screen "main" 1920x1080, template "Template_1"
   TextField "Static Text47_8" at 798,552 size 36x17; Text 'TE1.3 / TE04.1'
   Group "Group_10" at 795,569 size 82x26
   SymbolLibrary "Symbol library_115" at 1565,119 size 14x20
      Visibility <- "Di_1Ga01"
      Appearance <- "ViewLine_DB_Line24"
   SymbolLibrary "Symbol library_114" at 1552,129 size 27x27
      Visibility <- "Di_1Ga01"
      Appearance <- "ViewLine_DB_Line24"
   SymbolLibrary "Symbol library_113" at 1520,142 size 34x14
      Visibility <- "Di_1Ga01"
      Appearance <- "ViewLine_DB_Line24"
   SymbolLibrary "Symbol library_116" at 1565,120 size 14x57
      Visibility <- "Di_1Ga02"
      Appearance <- "ViewLine_DB_Line25"
   SymbolLibrary "Symbol library_117" at 1552,167 size 27x27
      Visibility <- "Di_1Ga02"
      Appearance <- "ViewLine_DB_Line25"
   SymbolLibrary "Symbol library_118" at 1520,180 size 34x14
      Visibility <- "Di_1Ga02"
      Appearance <- "ViewLine_DB_Line25"
   Rectangle "Rectangle_1r" at 50,206 size 75x24; ToolTipText 'Температура НС'
   TextField "Text field_1asd" at 100,206 size 19x22; Text 'С°'
   IOField "IO Field_10" at 43,204 size 56x26; FormatPattern 999.9
      ProcessValue <- "AiCh_TE7.1_Px"
   Rectangle "Rectangle_2cxv" at 182,511 size 75x24; ToolTipText 'Температура НС'
   TextField "Text field_3df" at 232,511 size 19x22; Text 'С°'
   IOField "IO Field_1" at 175,509 size 56x26; FormatPattern 999.9
      ProcessValue <- "AiCh_TE7.2_Px"
   Rectangle "Rectangle_3dcxf" at 920,570 size 75x24; ToolTipText 'Температура НС'
   TextField "Text field_4ыва" at 970,570 size 19x22; Text 'С°'
   IOField "IO Field_2" at 913,568 size 56x26; FormatPattern 999.9
      ProcessValue <- "AiCh_TE1.1_Px"
   Rectangle "Rectangle_4" at 921,495 size 68x24; ToolTipText 'Температура НС'
   TextField "Text field_6ret" at 962,495 size 18x22; Text '%'
   IOField "IO Field_3" at 924,493 size 36x26; FormatPattern 999
      ProcessValue <- "AiCh_LIC1.1_Px"
   Rectangle "Rectangle_5" at 802,571 size 75x24; ToolTipText 'Температура НС'
   IOField "IO Field_4" at 795,569 size 56x26; FormatPattern 999.9
      ProcessValue <- "AiCh_TE1.3_Px"
   TextField "Text field_8qw" at 852,571 size 19x22; Text 'С°'
   Rectangle "Rectangle_6" at 804,342 size 75x24; ToolTipText 'Температура НС'
   IOField "IO Field_5" at 797,340 size 56x26; FormatPattern 999.9
      ProcessValue <- "AiCh_TE1.2_Px"
   TextField "Text field_9x" at 854,342 size 19x22; Text 'С°'
   Rectangle "Rectangle_8" at 1342,495 size 68x24; ToolTipText 'Температура НС'
   TextField "Text field_11as" at 1383,495 size 18x22; Text '%'
   IOField "IO Field_6" at 1345,493 size 36x26; FormatPattern 999
      ProcessValue <- "AiCh_LIC2.1_Px"
   Rectangle "Rectangle_9" at 1341,570 size 75x24; ToolTipText 'Температура НС'
   TextField "Text field_12ew" at 1391,570 size 19x22; Text 'С°'
   IOField "IO Field_7" at 1334,568 size 56x26; FormatPattern 999.9
      ProcessValue <- "AiCh_TE2.1_Px"
   TextField "Static Text47_5" at 1219,547 size 36x17; Text 'TE2.3 / TE04.1'
   Group "Group_12" at 1216,564 size 82x26
   Rectangle "Rectangle_10" at 1223,566 size 75x24; ToolTipText 'Температура НС'
   IOField "IO Field_8" at 1216,564 size 56x26; FormatPattern 999.9
      ProcessValue <- "AiCh_TE2.3_Px"
   TextField "Text field_13azq" at 1273,566 size 19x22; Text 'С°'
   Group "Group_14" at 797,340 size 82x26
   TextField "Static Text47_7" at 820,324 size 36x17; Text 'TE1.2 / TE04.1'
   Rectangle "Rectangle_11" at 1225,342 size 75x24; ToolTipText 'Температура НС'
   IOField "IO Field_9" at 1218,340 size 56x26; FormatPattern 999.9
      ProcessValue <- "AiCh_TE2.2_Px"
   TextField "Text field_14ty" at 1275,342 size 19x22; Text 'С°'
   Group "Group_16" at 1218,340 size 82x26
   TextField "Static Text47_10" at 1241,324 size 36x17; Text 'TE2.2 / TE04.1'
   Rectangle "Rectangle_12" at 230,351 size 68x24; ToolTipText 'Температура НС'
   TextField "Text field_15fd" at 271,351 size 18x22; Text '%'
   IOField "IO Field_11" at 233,349 size 36x26; FormatPattern 999
      ProcessValue <- "Data.LevelVO"
   IOField "I/O field_2" at 165,649 size 39x20; FormatPattern 999
      ProcessValue <- "Data_Reg_01RV01_LMN"
   TextField "Text field_16d" at 201,650 size 19x19; Text '%'
   IOField "I/O field_1" at 309,929 size 39x20; FormatPattern 999
      ProcessValue <- "DriveM7_1.Vx"
   TextField "Text field_17zzz" at 345,930 size 19x19; Text '%'
   IOField "I/O field_3" at 562,932 size 39x20; FormatPattern 999
      ProcessValue <- "DriveM7_2.Vx"
   TextField "Text field_18" at 598,933 size 19x19; Text '%'
   IOField "I/O field_4" at 921,245 size 43x20; FormatPattern s999
      ProcessValue <- "DriveM1_1.Vx"
   TextField "Text field_19" at 965,246 size 19x19; Text '%'
   IOField "I/O field_6" at 1342,245 size 43x20; FormatPattern s999
      ProcessValue <- "DriveM2_1.Vx"
   TextField "Text field_21" at 1386,246 size 19x19; Text '%'
   Rectangle "Rectangle_13" at 182,487 size 75x24; ToolTipText 'Температура НС'
   TextField "Text field_20" at 232,487 size 19x22; Text 'С°'
   IOField "IO Field_17" at 175,485 size 56x26; FormatPattern 999.9
      ProcessValue <- "Data_Reg_01RV01_Sp"
   Rectangle "Rectangle_14" at 920,546 size 75x24; ToolTipText 'Температура НС'
   TextField "Text field_22" at 970,546 size 19x22; Text 'С°'
   IOField "IO Field_18" at 913,544 size 56x26; FormatPattern 999.9
      ProcessValue <- "Data_Reg_TE1_1_Sp"
   Rectangle "Rectangle_15" at 230,327 size 68x24; ToolTipText 'Температура НС'
   TextField "Text field_23" at 271,327 size 18x22; Text '%'
   IOField "IO Field_19" at 233,325 size 36x26; FormatPattern 999
      ProcessValue <- "Data_Reg_M7_1_Sp"
   Rectangle "Rectangle_16" at 1341,546 size 75x24; ToolTipText 'Температура НС'
   TextField "Text field_24" at 1391,546 size 19x22; Text 'С°'
   IOField "IO Field_20" at 1334,544 size 56x26; FormatPattern 999.9
      ProcessValue <- "Data_Reg_TE2_1_Sp"
   SymbolLibrary "Symbol library_130" at 703,869 size 202x14
      Appearance <- "ViewLine_DB_Line23"
   SymbolLibrary "Symbol library_15" at 917,869 size 415x14
      Appearance <- "ViewLine_DB_Line18"
   SymbolLibrary "Symbol library_49" at 1379,706 size 111x13
      Appearance <- "ViewLine_DB_Line17"
   SymbolLibrary "Symbol library_3" at 861,370 size 31x13
      Appearance <- "ViewLine_DB_Line11"
   SymbolLibrary "Symbol library_45" at 959,706 size 111x13
      Appearance <- "ViewLine_DB_Line13"
   SymbolLibrary "Symbol library_106" at 345,501 size 12x113
      Appearance <- "ViewLine_DB_Line7"
   SymbolLibrary "Symbol library_82" at 289,819 size 14x38
      Appearance <- "ViewLine_DB_Line3"
   SymbolLibrary "Symbol library_16" at 260,444 size 14x436
      Appearance <- "ViewLine_DB_Line1"
   SymbolLibrary "Symbol library_156" at 569,331 size 25x25
      Appearance <- "DrvCell_M3_Km1"
   SymbolLibrary "Symbol library_157" at 460,326 size 53x13
      Appearance <- "DrvCell_M3_Km1"
   ScreenModuleView "M_3_1" at 511,323 size 60x51; ScreenModuleType ""
      Guid_{11997190-24475} <- "DrvCell_M3_Err"
      Guid_{11997190-24471} <- "DrvCell_M3_Km1"
   Button "Button_4ert" at 510,323 size 61x52; TextOff 'Text'
      on Press: function_b14e0dd5("DrvCell_M3_SB1", 0)
   SymbolLibrary "Symbol library_44" at 949,604 size 14x235
      Appearance <- "ViewLine_DB_Line10"
   SymbolLibrary "Symbol library_66" at 885,598 size 25x25
      Appearance <- "ViewLine_DB_Line11"
   GraphicView "Graphic view_5" at 872,330 size 164x288; Picture "Graphic_1"
   SymbolLibrary "Symbol library_39" at 552,854 size 12x25
      Appearance <- "ViewLine_DB_Line4"
   SymbolLibrary "Symbol library_21" at 365,499 size 12x64
      Appearance <- "ViewLine_DB_Line6"
   SymbolLibrary "Symbol library_80" at 1586,695 size 96x14
      Appearance <- "ViewLine_DB_Line21"
   SymbolLibrary "Symbol library_14" at 214,202 size 25x25
      Appearance <- "ViewLine_DB_Line2"
   SymbolLibrary "Symbol library_10" at 153,224 size 13x158
      Appearance <- "ViewLine_DB_Line2"
   SymbolLibrary "Symbol library_47" at 107,377 size 125x14
      Appearance <- "ViewLine_DB_Line1"
   SymbolLibrary "Symbol library_5" at 218,206 size 98x241
   Bar "Bar_5" at 224,244 size 86x168; MinimumValue 0; MaximumValue 100
      ProcessValue <- "Data.LevelVO"
   SymbolLibrary "Symbol library_71" at 1306,598 size 25x25
      Appearance <- "ViewLine_DB_Line15"
   SymbolLibrary "Symbol library_56" at 1282,370 size 31x13
      Appearance <- "ViewLine_DB_Line15"
   SymbolLibrary "Symbol library_9" at 1369,604 size 14x235
      Appearance <- "ViewLine_DB_Line14"
   GraphicView "Graphic view_1" at 1293,330 size 164x288; Picture "Graphic_1"
   Bar "Bar_1" at 1314,352 size 124x243; MinimumValue 0; MaximumValue 100
      ProcessValue <- "AiCh_LIC2.1_Px"
   Bar "Bar_2" at 893,352 size 124x243; MinimumValue 0; MaximumValue 100
      ProcessValue <- "AiCh_LIC1.1_Px"
   SymbolLibrary "Symbol library_110" at 968,800 size 395x14
      Appearance <- "ViewLine_DB_Line3"
   SymbolLibrary "Symbol library_53" at 32,131 size 14x237
      Appearance <- "ViewLine_DB_Line1"
   SymbolLibrary "Symbol library_11" at 177,202 size 47x13
      Appearance <- "ViewLine_DB_Line2"
   SymbolLibrary "Symbol library_58" at 28,105 size 21x41
   SymbolLibrary "Symbol library_23" at 381,476 size 104x12
      Appearance <- "ViewLine_DB_Line5"
   SymbolLibrary "Symbol library_25" at 492,495 size 12x189
      Appearance <- "ViewLine_DB_Line5"
   SymbolLibrary "Symbol library_79" at 381,440 size 140x12
      Appearance <- "ViewLine_DB_Line4"
   SymbolLibrary "Symbol library_6" at 253,150 size 54x59
   SymbolLibrary "Symbol library_7" at 303,150 size 65x30
   SymbolLibrary "Symbol library_158" at 581,299 size 13x35
      Appearance <- "DrvCell_M3_Km1"
   SymbolLibrary "Symbol library_160" at 578,147 size 13x58
   SymbolLibrary "Symbol library_31" at 284,885 size 31x16
   SymbolLibrary "Symbol library_36" at 1335,869 size 156x14
      Appearance <- "ViewLine_DB_Line19"
   SymbolLibrary "Symbol library_12" at 153,202 size 25x25
      Appearance <- "ViewLine_DB_Line2"
   TextField "Text field_2fdsa" at 314,702 size 19x34; Text 'Y'
   SymbolLibrary "Symbol library_186" at 678,132 size 14x727
      Appearance <- "ViewLine_DB_Line23"
   SymbolLibrary "Symbol library_41" at 271,906 size 15x15
      Appearance <- "ViewLine_DB_Line8"
   SymbolLibrary "Symbol library_46" at 168,934 size 99x8
      Appearance <- "ViewLine_DB_Line8"
   SymbolLibrary "Symbol library_43" at 146,930 size 30x15
   SymbolLibrary "Symbol library_48" at 264,927 size 15x15
      Appearance <- "ViewLine_DB_Line8"
   SymbolLibrary "Symbol library_50" at 271,914 size 8x16
      Appearance <- "ViewLine_DB_Line8"
   SymbolLibrary "Symbol library_95" at 678,107 size 27x27
      Appearance <- "ViewLine_DB_Line23"
   SymbolLibrary "Symbol library_91" at 1012,142 size 503x14
      Appearance <- "ViewLine_DB_Line24"
   SymbolLibrary "Symbol library_90" at 693,107 size 824x14
      Appearance <- "ViewLine_DB_Line23"
   SymbolLibrary "Symbol library_93" at 1439,180 size 78x14
      Appearance <- "ViewLine_DB_Line25"
   SymbolLibrary "Symbol library_98" at 1577,107 size 293x14
      Appearance <- "ViewLine_DB_Line22"
   SymbolLibrary "Symbol library_99" at 574,121 size 21x41
   SymbolLibrary "Symbol library_100" at 442,321 size 41x21
   SymbolLibrary "Symbol library_108" at 1590,546 size 95x14
      Appearance <- "ViewLine_DB_Line20"
   SymbolLibrary "Symbol library_109" at 1672,542 size 41x21
   SymbolLibrary "Symbol library_107" at 313,800 size 211x14
      Appearance <- "ViewLine_DB_Line3"
   SymbolLibrary "Symbol library_111" at 1388,800 size 105x14
      Appearance <- "ViewLine_DB_Line3"
   SymbolLibrary "Symbol library_105" at 1479,796 size 41x21
   TextField "Static Text47_2" at 199,470 size 33x16; Text 'TE7.2 / TE04.1'
   SymbolLibrary "Symbol library_29" at 695,800 size 247x14
      Appearance <- "ViewLine_DB_Line3"
   Circle "Circle_23" at 1030,351 size 25x25
      Appearance <- "Di_Lah1.1"
   SymbolLibrary "Symbol library_57" at 944,610 size 37x48
   TextField "Static Text47_6" at 938,530 size 33x16; Text 'TE1.1 / TE04.1'
   TextField "Static Text47_9" at 935,479 size 40x16; Text 'LIC 1.1 / TE04.1'
   SymbolLibrary "Symbol library_123" at 989,168 size 14x209
      Appearance <- "ViewLine_DB_Line24"
   SymbolLibrary "Symbol library_55" at 989,142 size 27x27
      Appearance <- "ViewLine_DB_Line24"
   SymbolLibrary "Symbol library_96" at 1415,180 size 27x27
      Appearance <- "ViewLine_DB_Line25"
   SymbolLibrary "Symbol library_97" at 678,856 size 27x27
      Appearance <- "ViewLine_DB_Line23"
   SymbolLibrary "Symbol library_83" at 289,800 size 27x27
      Appearance <- "ViewLine_DB_Line3"
   SymbolLibrary "Symbol library_18" at 260,874 size 27x27
      Appearance <- "ViewLine_DB_Line1"
   SymbolLibrary "Symbol library_54" at 32,364 size 27x27
      Appearance <- "ViewLine_DB_Line1"
   SymbolLibrary "Symbol library_24" at 480,476 size 24x22
      Appearance <- "ViewLine_DB_Line5"
   GraphicView "Graphic view_4" at 526,196 size 122x112; Picture "Graphic_5"
   Circle "Circle_26" at 617,208 size 25x25
      Appearance <- "Di_Lah01"
   Circle "Circle_15" at 617,271 size 25x25
      Appearance <- "Di_Lal01"
   Line "Line_3" at 913,810 size 42x26
      Visibility <- "Di_Ga1.1"
   Line "Line_5" at 1333,810 size 42x26
      Visibility <- "Di_Ga2.1"
   Line "Line_1" at 913,838 size 42x36
      Visibility <- "Di_Ga1.2"
   Line "Line_6" at 1333,838 size 42x36
      Visibility <- "Di_Ga2.2"
   SymbolLibrary "Symbol library_94" at 1516,107 size 50x14
      Visibility <- "Di_1Ga06"
      Appearance <- "ViewLine_DB_Line23"
   Group "Group_2" at 1520,119 size 59x37
      Visibility <- "Di_1Ga01"
   Group "Group_3" at 1520,120 size 59x74
      Visibility <- "Di_1Ga02"
   ScreenModuleView "V7_31_2" at 76,350 size 50x42; ScreenModuleType ""
      Guid_{11997190-20001} <- "DrvCell_V7_3_Err"
      Guid_{11997190-19997} <- "DrvCell_V7_3_Km1"
   TextField "Static Text47_1" at 68,190 size 33x16; Text 'TE7.1 / TE04.1'
   Group "Group_17" at 43,204 size 82x26; FormatPattern 999.9
   Group "Group_1" at 175,509 size 82x26; FormatPattern 999.9
   ScreenModuleView "M7_1_1" at 283,856 size 88x65; ScreenModuleType ""
      Guid_{11997190-20935} <- "DrvCell_M7_1_Km1"
      Guid_{11997190-20939} <- "DrvCell_M7_1_Err"
   ScreenModuleView "M1_2_3" at 1480,850 size 60x51; ScreenModuleType ""
      Guid_{11997190-21672} <- "DrvCell_M5_Err"
      Guid_{11997190-21676} <- "DrvCell_M5_Km1"
   SymbolLibrary "Symbol library_17" at 910,338 size 88x135
   ScreenModuleView "M1_1_1" at 923,270 size 53x69; ScreenModuleType ""
      Guid_{11997190-22971} <- "DrvCell_M1_1_Err"
      Guid_{11997190-22975} <- "DrvCell_M1_1_Km1"
   SymbolLibrary "Symbol library_13" at 1364,610 size 37x48
   SymbolLibrary "Symbol library_92" at 1415,202 size 14x173
      Appearance <- "ViewLine_DB_Line25"
   SymbolLibrary "Symbol library_33" at 1333,338 size 88x135
   ScreenModuleView "M1_1_2" at 1347,270 size 53x69; ScreenModuleType ""
      Guid_{11997190-22971} <- "DrvCell_M2_1_Err"
      Guid_{11997190-22975} <- "DrvCell_M2_1_Km1"
   TextField "Text field_10v" at 1308,367 size 55x39; Text '№2'
   ScreenModuleView "V1_7_1" at 992,696 size 35x26; ScreenModuleType ""
      Guid_{11997190-23352} <- "DrvCell_V1_7_Err"
      Guid_{11997190-23356} <- "DrvCell_V1_7_Km1"
   Group "Group_6" at 921,493 size 68x26
   Group "Group_7" at 913,568 size 82x26
   TextField "Static Text47_3" at 1359,530 size 33x16; Text 'TE2.1 / TE04.1'
   TextField "Static Text47_4" at 1356,479 size 40x16; Text 'LIC 2.1 / TE04.1'
   Group "Group_8" at 1342,493 size 68x26
   Group "Group_9" at 1334,568 size 82x26
   Circle "Circle_3" at 1451,352 size 25x25
      Appearance <- "Di_Lah2.1"
   SymbolLibrary "Symbol library_67" at 838,370 size 25x25
      Appearance <- "ViewLine_DB_Line11"
   SymbolLibrary "Symbol library_147" at 814,390 size 25x25
      Appearance <- "ViewLine_DB_Line11"
   SymbolLibrary "Symbol library_102" at 814,413 size 13x26
      Appearance <- "ViewLine_DB_Line11"
   SymbolLibrary "Symbol library_64" at 838,393 size 13x257
      Appearance <- "ViewLine_DB_Line11"
   SymbolLibrary "Symbol library_65" at 906,610 size 25x25
      Appearance <- "ViewLine_DB_Line11"
   SymbolLibrary "Symbol library_63" at 906,622 size 25x25
      Appearance <- "ViewLine_DB_Line11"
   SymbolLibrary "Symbol library_59" at 738,649 size 114x13
      Appearance <- "ViewLine_DB_Line12"
   SymbolLibrary "Symbol library_68" at 708,645 size 41x21
   ScreenModuleView "V7_31_1" at 772,621 size 50x42; ScreenModuleType ""
      Guid_{11997190-20001} <- "DrvCell_V1_1_Err"
      Guid_{11997190-19997} <- "DrvCell_V1_1_Km1"
   SymbolLibrary "Symbol library_101" at 810,422 size 21x41
   SymbolLibrary "Symbol library_60" at 1259,370 size 25x25
      Appearance <- "ViewLine_DB_Line15"
   SymbolLibrary "Symbol library_61" at 1235,390 size 25x25
      Appearance <- "ViewLine_DB_Line15"
   SymbolLibrary "Symbol library_69" at 1235,413 size 13x26
      Appearance <- "ViewLine_DB_Line15"
   SymbolLibrary "Symbol library_70" at 1259,393 size 13x257
      Appearance <- "ViewLine_DB_Line15"
   SymbolLibrary "Symbol library_73" at 1327,610 size 25x25
      Appearance <- "ViewLine_DB_Line15"
   SymbolLibrary "Symbol library_74" at 1327,622 size 25x25
      Appearance <- "ViewLine_DB_Line15"
   SymbolLibrary "Symbol library_75" at 1159,649 size 114x13
      Appearance <- "ViewLine_DB_Line16"
   SymbolLibrary "Symbol library_76" at 1129,645 size 41x21
   SymbolLibrary "Symbol library_62" at 1231,422 size 21x41
   ScreenModuleView "V7_31_3" at 1196,621 size 50x42; ScreenModuleType ""
      Guid_{11997190-20001} <- "DrvCell_V2_1_Err"
      Guid_{11997190-19997} <- "DrvCell_V2_1_Km1"
   ScreenModuleView "V1_7_2" at 1412,696 size 35x26; ScreenModuleType ""
      Guid_{11997190-23352} <- "DrvCell_V2_7_Err"
      Guid_{11997190-23356} <- "DrvCell_V2_7_Km1"
   Group "Group_19" at 230,349 size 68x26
   ScreenModuleView "V1_7_3" at 198,923 size 35x26; ScreenModuleType ""
      Guid_{11997190-23352} <- "DrvCell_V7_1_Err"
      Guid_{11997190-23356} <- "DrvCell_V7_1_Km1"
   TextField "Static Text47_11" at 82,330 size 26x16; Text 'V7.3 / TE04.1'
   TextField "Static Text47_12" at 179,234 size 26x16; Text 'V7.4 / TE04.1'
   Button "Button_1yt" at 75,350 size 52x43; TextOff 'Text'
      on Press: function_b14e0dd5("DrvCell_V7_3_SB1", 0)
   SymbolLibrary "Symbol library_42" at 441,695 size 52x12
      Appearance <- "ViewLine_DB_Line5"
   SymbolLibrary "Symbol library_30" at 339,679 size 45x12
      Appearance <- "ViewLine_DB_Line5"
   ScreenModuleView "M_3_2" at 382,676 size 60x51; ScreenModuleType ""
      Guid_{11997190-24471} <- "DrvCell_M10_Km1"
      Guid_{11997190-24475} <- "DrvCell_M10_Err"
   SymbolLibrary "Symbol library_27" at 528,459 size 12x422
      Appearance <- "ViewLine_DB_Line4"
   SymbolLibrary "Symbol library_1" at 481,683 size 23x24
      Appearance <- "ViewLine_DB_Line5"
   SymbolLibrary "Symbol library_22" at 516,440 size 24x22
      Appearance <- "ViewLine_DB_Line4"
   SymbolLibrary "Symbol library_34" at 528,875 size 23x23
      Appearance <- "ViewLine_DB_Line4"
   SymbolLibrary "Symbol library_40" at 318,679 size 23x23
      Appearance <- "ViewLine_DB_Line5"
   TextField "adasd" at 650,858 size 19x34; Text 'Y'
   TextField "Static Text47_13" at 393,659 size 24x16; Text 'M10 / TE04.1'
   Button "Button_3fdg" at 382,676 size 60x52; TextOff 'Text'
      on Press: function_b14e0dd5("DrvCell_M10_SB1", 0)
   TextField "Static Text47_14" at 526,306 size 17x16; Text 'M3 / TE04.1'
   SymbolLibrary "Symbol library_2" at 361,550 size 21x41
   SymbolLibrary "Symbol library_19" at 643,834 size 23x23
      Appearance <- "ViewLine_DB_Line4"
   SymbolLibrary "Symbol library_20" at 573,834 size 76x12
      Appearance <- "ViewLine_DB_Line4"
   SymbolLibrary "Symbol library_26" at 552,834 size 23x23
      Appearance <- "ViewLine_DB_Line4"
   SymbolLibrary "Symbol library_28" at 533,912 size 8x22
      Appearance <- "ViewLine_DB_Line9"
   SymbolLibrary "Symbol library_32" at 526,927 size 15x15
      Appearance <- "ViewLine_DB_Line9"
   SymbolLibrary "Symbol library_37" at 533,899 size 15x15
      Appearance <- "ViewLine_DB_Line9"
   SymbolLibrary "Symbol library_38" at 444,934 size 87x8
      Appearance <- "ViewLine_DB_Line9"
   ScreenModuleView "V1_7_4" at 473,923 size 35x26; ScreenModuleType ""
      Guid_{11997190-23352} <- "DrvCell_V7_2_Err"
      Guid_{11997190-23356} <- "DrvCell_V7_2_Km1"
   TextField "Static Text58_1" at 9,65 size 62x32; Text 'Продукт, CIP+2 RV01'
   TextField "Static Text58_3" at 1474,770 size 35x16; Text 'CIP-2 / RV01'
   TextField "Static Text58_5" at 1716,535 size 62x32; Text 'Продукт, CIP+1 RV01'
   TextField "Static Text47_15" at 328,854 size 28x16; Text 'M7.1 / TE04.1'
   TextField "Static Text47_16" at 577,856 size 28x16; Text 'M7.2 / TE04.1'
   TextField "Static Text47_17" at 202,902 size 26x16; Text 'V7.1 / TE04.1'
   TextField "Static Text47_18" at 777,602 size 26x16; Text 'V1.1 / TE04.1'
   TextField "Static Text47_19" at 855,609 size 28x16; Text 'M1.2 / TE04.1'
   TextField "Static Text47_20" at 995,677 size 26x16; Text 'V1.7 / TE04.1'
   TextField "Static Text47_21" at 935,228 size 28x16; Text 'M1.1 / TE04.1'
   TextField "Static Text47_22" at 1359,228 size 28x16; Text 'M2.1 / TE04.1'
   TextField "Static Text47_23" at 1200,602 size 26x16; Text 'V2.1 / TE04.1'
   TextField "Static Text47_24" at 1276,609 size 28x16; Text 'M2.2 / TE04.1'
   TextField "Static Text47_25" at 1416,677 size 26x16; Text 'V2.7 / TE04.1'
   Button "Button_15" at 1398,684 size 65x49; TextOff 'Text'
      on Press: function_b14e0dd5("DrvCell_V2_7_SB1", 0)
   TextField "Static Text47_26" at 477,904 size 26x16; Text 'V7.2 / TE04.1'
   TextField "Static Text47_27" at 1785,887 size 17x16; Text 'M4 / TE04.1'
   TextField "Text field_7fd" at 885,367 size 55x39; Text '№1'
   Group "Group_11" at 795,552 size 82x43
   Group "Group_15" at 797,324 size 82x42
   Group "Group_18" at 1218,324 size 82x42
   Group "Group_13" at 1216,547 size 82x43; Text 'TE1.3'
   TextField "Static Text58_6" at 554,230 size 67x32; Text 'Ледянная вода RV01'
   TextField "Static Text58_7" at 81,922 size 61x32; Text 'Вода питьевая RV01'
   SymbolLibrary "Symbol library_35" at 1575,566 size 14x288
      Appearance <- "ViewLine_DB_Line20"
   SymbolLibrary "Symbol library_72" at 1540,853 size 35x14
      Appearance <- "ViewLine_DB_Line20"
   SymbolLibrary "Symbol library_77" at 1562,840 size 27x27
      Appearance <- "ViewLine_DB_Line20"
   SymbolLibrary "Symbol library_78" at 1575,546 size 27x27
      Appearance <- "ViewLine_DB_Line20"
   SymbolLibrary "Symbol library_81" at 1690,708 size 14x66
      Appearance <- "ViewLine_DB_Line21"
   SymbolLibrary "Symbol library_84" at 1677,695 size 27x27
      Appearance <- "ViewLine_DB_Line21"
   SymbolLibrary "Symbol library_85" at 1690,865 size 14x50
      Appearance <- "ViewLine_DB_Line21"
   SymbolLibrary "Symbol library_86" at 1707,926 size 55x14
      Appearance <- "ViewLine_DB_Line21"
   SymbolLibrary "Symbol library_87" at 1690,913 size 27x27
      Appearance <- "ViewLine_DB_Line21"
   GraphicView "Graphic view_2" at 1636,758 size 122x112; Picture "Graphic_5"
   TextField "Static Text58_4" at 1687,789 size 21x32; Text 'CIP ББ RV01'
   SymbolLibrary "Symbol library_88" at 1869,123 size 14x788
      Appearance <- "ViewLine_DB_Line22"
   SymbolLibrary "Symbol library_89" at 1818,910 size 48x14
      Appearance <- "ViewLine_DB_Line22"
   SymbolLibrary "Symbol library_103" at 1856,897 size 27x27
      Appearance <- "ViewLine_DB_Line22"
   SymbolLibrary "Symbol library_51" at 1856,107 size 27x27
      Appearance <- "ViewLine_DB_Line22"
   TextField "Static Text47_28" at 1503,830 size 17x16; Text 'M5 / TE04.1'
   ScreenModuleView "M1_2_4" at 1759,906 size 60x51; ScreenModuleType ""
      Guid_{11997190-21672} <- "DrvCell_M4_Err"
      Guid_{11997190-21676} <- "DrvCell_M4_Km1"
   SymbolLibrary "Symbol library_104" at 543,800 size 131x14
      Appearance <- "ViewLine_DB_Line3"
   SymbolLibrary "Symbol library_112" at 277,624 size 63x12
      Appearance <- "ViewLine_DB_Line7"
   SymbolLibrary "Symbol library_119" at 128,625 size 128x12
      Appearance <- "ViewLine_DB_Line7"
   SymbolLibrary "Symbol library_120" at 334,612 size 23x24
      Appearance <- "ViewLine_DB_Line7"
   SymbolLibrary "Symbol library_121" at 107,638 size 12x105
      Appearance <- "ViewLine_DB_Line7"
   SymbolLibrary "Symbol library_122" at 107,625 size 22x22
      Appearance <- "ViewLine_DB_Line7"
   SymbolLibrary "Symbol library_124" at 102,736 size 21x41
   Group "Group_20" at 165,649 size 55x20; FormatPattern 999
   Group "Group_21" at 309,929 size 55x20; FormatPattern 999
   Group "Group_22" at 562,932 size 55x20; FormatPattern 999
   Group "Group_23" at 921,245 size 63x20; FormatPattern 999
   Group "Group_25" at 1342,245 size 63x20; FormatPattern 999
   SymbolLibrary "Symbol library_127" at 1298,286 size 41x32
      Visibility <- "Data_Mixer2_Direction"
   SymbolLibrary "Symbol library_128" at 1414,286 size 41x32
      Visibility <- "Data_Mixer2_Direction"
   TextField "Text field_68" at 562,60 size 776x42; Text 'Активный ручной режим'
      Visibility <- "Data_MAN_ON"
   Button "Button_13vf" at 1186,619 size 65x54; TextOff 'Text'
      on Press: function_b14e0dd5("DrvCell_V2_1_SB1", 0)
   IOField "IO Field_12" at 106,587 size 47x31; FormatPattern 999
      ProcessValue <- "Data_Reg_01RV01_Man"
      Visibility <- "Data_MAN_ON"
   ScreenModuleView "RV01_1" at 157,579 size 51x64; ScreenModuleType ""
      Guid_{11997190-34850} <- "Data_Reg_01RV01_LMN"
   IOField "IO Field_13" at 373,919 size 47x31; FormatPattern 999
      Visibility <- "Data_MAN_ON"
      ProcessValue <- "Data_Reg_M7_1_Man"
   IOField "IO Field_14" at 626,919 size 47x31; FormatPattern 999
      Visibility <- "Data_MAN_ON"
      ProcessValue <- "Data_Reg_M7_2_Man"
   IOField "IO Field_15" at 859,244 size 51x31; FormatPattern s999
      Visibility <- "Data_MAN_ON"
      ProcessValue <- "Data_Mixer1_Man"
   IOField "IO Field_16" at 1284,244 size 51x31; FormatPattern s999
      Visibility <- "Data_MAN_ON"
      ProcessValue <- "Data_Mixer2_Man"
   Button "Button_18" at 1474,838 size 72x71; TextOff 'Text'
      on Press: function_b14e0dd5("DrvCell_M5_SB1", 0)
   Button "Button_17" at 1753,894 size 72x71; TextOff 'Text'
      on Press: function_b14e0dd5("DrvCell_M4_SB1", 0)
   SymbolLibrary "Symbol library_164" at 872,286 size 41x32
      Visibility <- "Data_Mixer1_Direction"
   SymbolLibrary "Symbol library_126" at 988,286 size 41x32
      Visibility <- "Data_Mixer1_Direction"
   Button "Button_12" at 914,266 size 74x78; TextOff 'Text'
      on Press: function_b14e0dd5("DrvCell_M1_1_SB1", 0)
   Group "Group_24" at 175,485 size 82x26; FormatPattern 999.9
   Group "Group_26" at 913,544 size 82x26
   Group "Group_27" at 230,325 size 68x26; FormatPattern 999
   Group "Group_28" at 1334,544 size 82x26
   Rectangle "Rectangle_17" at 905,346 size 20x20
      Appearance <- "Di_Ga1.4"
   Rectangle "Rectangle_18" at 1327,346 size 20x20
      Appearance <- "Di_Ga2.4"
   SymbolLibrary "Symbol library_125" at 427,930 size 30x15
   Button "Button_9" at 472,922 size 37x27; TextOff 'Text'
      on Press: function_b14e0dd5("DrvCell_V7_2_SB1", 0)
   Button "Button_8" at 197,921 size 36x29; TextOff 'Text'
      on Press: function_b14e0dd5("DrvCell_V7_1_SB1", 0)
   Button "Button_6asd" at 762,619 size 65x49; TextOff 'Text'
      on Press: function_b14e0dd5("DrvCell_V1_1_SB1", 0)
   Button "Button_11" at 977,684 size 65x49; TextOff 'Text'
      on Press: function_b14e0dd5("DrvCell_V1_7_SB1", 0)
   ScreenModuleView "M7_21_1" at 547,869 size 77x60; ScreenModuleType ""
      Guid_{11997190-26153} <- "DrvCell_M7_2_Err"
      Guid_{11997190-26157} <- "DrvCell_M7_2_Km1"
   Button "Button_7" at 545,869 size 80x61; TextOff 'Text'
      on Press: function_b14e0dd5("DrvCell_M7_2_SB1", 0)
   ScreenModuleView "М7_4_1" at 151,259 size 42x50; ScreenModuleType ""
      Guid_{11997190-20546} <- "DrvCell_V7_4_Err"
      Guid_{11997190-20554} <- "DrvCell_V7_4_Km1"
   Button "Button_2xz" at 151,257 size 42x52; TextOff 'Text'
      on Press: function_b14e0dd5("DrvCell_V7_4_SB1", 0)
   SymbolLibrary "Symbol library_129" at 55,377 size 22x14
      Appearance <- "ViewLine_DB_Line1"
   SymbolLibrary "Symbol library_4" at 1059,701 size 41x21
   SymbolLibrary "Symbol library_132" at 838,637 size 25x25
      Appearance <- "ViewLine_DB_Line11"
   ScreenModuleView "M1_2_1" at 854,629 size 60x51; ScreenModuleType ""
      Guid_{11997190-21672} <- "DrvCell_M1_2_Err"
      Guid_{11997190-21676} <- "DrvCell_M1_2_Km1"
   Button "Button_10" at 848,623 size 74x64; TextOff 'Text'
      on Press: function_b14e0dd5("DrvCell_M1_2_SB1", 0)
   Button "Button_5r" at 282,855 size 90x67; TextOff 'Text'
      on Press: function_b14e0dd5("DrvCell_M7_1_SB1", 0)
   SymbolLibrary "Symbol library_52" at 1479,701 size 41x21
   SymbolLibrary "Symbol library_131" at 1259,637 size 25x25
      Appearance <- "ViewLine_DB_Line15"
   ScreenModuleView "M1_2_2" at 1275,629 size 60x51; ScreenModuleType ""
      Guid_{11997190-21672} <- "DrvCell_M2_2_Err"
      Guid_{11997190-21676} <- "DrvCell_M2_2_Km1"
   Button "Button_14" at 1267,623 size 74x64; TextOff 'Text'
      on Press: function_b14e0dd5("DrvCell_M2_2_SB1", 0)
   SymbolLibrary "Symbol library_8" at 339,116 size 43x399
   Button "Button_16" at 1338,266 size 74x78; TextOff 'Text'
      on Press: function_b14e0dd5("DrvCell_M2_1_SB1", 0)
   TextField "Static Text47_29" at 167,557 size 30x16; Text 'RV01 / TE04.1'
   TextField "Static Text47_30" at 733,745 size 42x16; Text 'Привет / TE04.1'

screen "settingsKr1" 1920x1080, template "Template_1"
   on GenerateScreen: SetTag("Tag_ScreenNumber", 8)
   TextField "Template_Text field_7" at 302,77 size 446x37; Text 'Параметры кристализации №1'
   TextField "Template_Text field_1" at 1184,77 size 360x37; Text 'Параметры мешалки №1'
   SymbolicIOField "Symbolic I/O field_kr1" at 272,432 size 506x55; TextOn '1'; TextOff '0'; TextList "Kristal_Regim"
      ProcessValue <- "Data_Kr1_Regim"
      ObjectEnable <- "Kr_1_Work_Run"
   TextField "Text field_12vxio" at 431,584 size 231x25; Text 'Готовность к включению'
   Circle "read_work_kr1" at 366,572 size 48x48
      Appearance <- "Data_Kr1_Ready_Work"
   Button "Button_1123" at 537,493 size 241x55; TextOff 'Стоп'
      on Press: function_b14e0dd5("Data_Kr1_Stop", 0)
   Button "Button_2123" at 272,493 size 241x55; TextOff 'Старт'
      on Press: function_b14e0dd5("Data_Kr1_Start", 0)
   TextField "Text field_1kr1" at 460,644 size 155x25; Text 'Маршрут собран'
   Circle "ready_route_kr1" at 403,636 size 40x40
      Appearance <- "Data_Kr1_Ready_Route"
   Circle "Circl_11" at 403,693 size 40x40
      Appearance <- "Data_MAN_ON"
   TextField "Text field_kr1" at 460,701 size 214x25; Text 'Режим автоматический'
   Group "Group_3" at 235,252 size 595x42
   Group "Group_4" at 235,304 size 595x42
   Group "Group" at 235,147 size 595x42
   Group "Group_2" at 235,199 size 595x42
   Circle "Circl_8" at 403,750 size 40x40
      Appearance <- "Data_ReadyKr1"
   TextField "Text field_2kr1" at 460,758 size 114x25; Text 'Разрешение'
   Group "Group_6" at 1048,147 size 594x42
   Group "Group_7" at 1048,199 size 594x42
   Group "Group_8" at 1048,252 size 594x42
   Group "Group_9" at 1048,304 size 594x42
   TextField "Template_Text field_6" at 1048,371 size 160x29; Text 'Режим мешалки'
   Button "Button_9" at 1392,358 size 118x55; TextOff '<< || >>'
      on Release: SetBit("Data_Mixer1_RegimBothSide")
      Appearance <- "Data_Mixer1_RegimBothSide"
   Button "Button_10" at 1524,358 size 118x55; TextOff '>>'
      on Release: ResetBit("Data_Mixer1_RegimBothSide")
      Appearance <- "Data_Mixer1_RegimBothSide"
   Group "Group_10" at 1148,433 size 431x55
   Button "Template_Button_1" at 1148,433 size 210x55; TextOff 'Старт мешалки'
      on Press: function_b14e0dd5("Data_Mixer1_Start", 0)
   Button "Template_Button_2" at 1369,433 size 210x55; TextOff 'Стоп мешалки'
      on Press: function_b14e0dd5("Data_Mixer1_Stop", 0)
   IOField "IO Field_15" at 1568,147 size 74x42; FormatPattern 999
      ProcessValue <- "Data_Mixer1_Power"
   TextField "Template_Text field_2" at 1048,154 size 217x29; Text 'Обороты мешалки, %'
   IOField "IO Field_1" at 1568,199 size 74x42; FormatPattern 9999
      ProcessValue <- "Data_Mixer1_TimeRight"
   TextField "Template_Text field_3" at 1048,206 size 288x29; Text 'Время вращения вправо, сек'
   IOField "IO Field_2" at 1568,252 size 74x42; FormatPattern 9999
      ProcessValue <- "Data_Mixer1_TimeLeft"
   TextField "Template_Text field_4" at 1048,259 size 276x29; Text 'Время вращения влево, сек'
   IOField "IO Field_3" at 1568,304 size 74x42; FormatPattern 9999
      ProcessValue <- "Data_Mixer1_TimePause"
   TextField "Template_Text field_5" at 1048,311 size 222x29; Text 'Время паузы мешалки'
   IOField "IO Field_4" at 756,147 size 74x42; FormatPattern 999.9
      ProcessValue <- "Data_Kr1_TempFilling"
      ObjectEnable <- "Kr_1_Work_Run"
   TextField "Template_Text field_8" at 235,154 size 289x29; Text 'Температура наполнения, С°'
   IOField "IO Field_5" at 756,199 size 74x42; FormatPattern 999.9
      ProcessValue <- "Data_Kr1_TempKristal"
      ObjectEnable <- "Kr_1_Work_Run"
   TextField "Template_Text field_9" at 235,206 size 319x29; Text 'Температура кристализации, С°'
   IOField "IO Field_6" at 756,252 size 74x42; FormatPattern 9999
      ProcessValue <- "Data_Kr1_TimeKristal"
      ObjectEnable <- "Kr_1_Work_Run"
   TextField "Template_Text field_10" at 235,259 size 268x29; Text 'Время кристализации, мин'
   IOField "IO Field_7" at 756,304 size 74x42; FormatPattern 999
      ProcessValue <- "Kr_1_Work_LeftTimeMin"
   TextField "Template_Text field_11" at 235,311 size 296x29; Text 'До конца кристализации, мин'

Template "Template_1" 1920x1080
   DateTimeField "Template_Date/time field_1" at 1793,0 size 120x30
   TextField "Text field_69" at 866,1 size 277x47; Text 'Работает кристализатор № 1'
      Visibility <- "Kr_1_Work_Run"
   TextField "Text field_10" at 1422,1 size 277x47; Text 'Мойка'
      Visibility <- "WashingWork_DB_Run"
   GraphicView "Graphic view_3" at 2,1 size 182x49; Picture "Graphic_2"
   Button "Button_13" at 120,1020 size 200x40; TextOff 'Главный экран'
      on Release: ActivateScreen("main", 0)
   Button "Button_1" at 340,1020 size 200x40; TextOff 'Графики'
      on Release: ActivateScreen("TrendsCommon", 0)
   Button "Button_2" at 560,1020 size 200x40; TextOff 'Сообщения'
      on Release: ActivateScreen("messages", 0)
   Button "Button_3" at 780,1020 size 200x40; TextOff 'Настройки'
      on Release: ActivateScreen("settingsCommon", 0)
   Button "Button_4" at 1000,1020 size 200x40; TextOff 'Сброс аварии'
      on Press: function_b14e0dd5("Data_ACK", 0)
   Button "Button_5" at 6,1001 size 96x70; TextOff 'Главный экран'; PictureOff "Arrow Left (1)"
      on Press: function_efd93a16()
   AlarmView "Template_Alarm view_1" at 0,973 size 1920x26
   Button "Button_6" at 1220,1020 size 200x40; TextOff 'Ручной'
      on Press: InvertBit("Data_MAN_ON")
      ObjectEnable <- "Data_Equipment_Work"
   TextField "Text field_9" at 1144,1 size 277x47; Text 'Работает кристализатор № 2'
      Visibility <- "Kr_2_Work_Run"
   TextField "Text field_14" at 1701,1 size 89x47; Text 'Ошибка'
      Visibility <- "Data_GlobalError"
   TextField "Text field_15" at 866,1 size 833x47; Text 'Аварийный останов'
      Visibility <- "Data_GlobalErrorStop"
   TextField "Text field_2" at 217,2 size 167x25; Text 'Режим крист. №1'
   TextField "Text field_1" at 247,23 size 107x23; Text 'Наполнение'
      Visibility <- "Kr_1_Work_Step"
   TextField "Text field_3" at 235,23 size 132x23; Text 'Кристализация'
      Visibility <- "Kr_1_Work_Step"
   TextField "Text field_4" at 262,23 size 79x23; Text 'Выкачка'
      Visibility <- "Kr_1_Work_Step"
   TextField "Text field_5" at 451,2 size 162x25; Text 'Режим крист. №2'
   TextField "Text field_6" at 479,23 size 107x23; Text 'Наполнение'
      Visibility <- "Kr_2_Work_Step"
   TextField "Text field_7" at 467,23 size 132x23; Text 'Кристализация'
      Visibility <- "Kr_2_Work_Step"
   TextField "Text field_8" at 494,23 size 79x23; Text 'Выкачка'
      Visibility <- "Kr_2_Work_Step"
   TextField "Text field_11" at 709,1 size 97x25; Text 'CIP Мойка'
   TextField "Text field_12" at 682,24 size 152x23; Text 'Подача продукта'
      Visibility <- "WashingWork_DB_Step"
   TextField "Text field_13" at 674,24 size 168x23; Text 'Выгрузка продукта'
      Visibility <- "WashingWork_DB_Step"
   TextField "Text field_16" at 714,24 size 88x23; Text 'Крист №1'
      Visibility <- "WashingWork_DB_Step"
   TextField "Text field_17" at 714,24 size 88x23; Text 'Крист №2'
      Visibility <- "WashingWork_DB_Step"
   DateTimeField "Template_Date/time field_2" at 1795,22 size 117x30

screen "messages" 1920x1080, template "Template_1"
   AlarmView "Alarm view_1" at 0,50 size 960x922
   AlarmView "Alarm view_2" at 960,50 size 960x922; ColumnTextNumber 'No. / №'; ColumnTextTime 'Time / Время'; ColumnTextAlarmState 'Status / Статус'; ColumnTextAlarmText 'Text / Текст'; ColumnTextDate 'Date / Дата'; ColumnTextAckGroup 'Acknowledge group / Квитировать группу'; ColumnTextDevice 'PLC / ПЛК'; AlarmLog "Alarm_log_1"

screen "Kristal_2" 1920x1080, template "Template_1"
   on GenerateScreen: SetTag("Tag_ScreenNumber", 6)
   TrendView "Trend view_1" at 0,51 size 1920x920

screen "Kristal_1" 1920x1080, template "Template_1"
   on GenerateScreen: SetTag("Tag_ScreenNumber", 5)
   TrendView "Trend view_1" at 0,51 size 1920x920

screen "TrendsCommon" 1920x1080, template "Template_1"
   on GenerateScreen: SetTag("Tag_ScreenNumber", 2)
   Button "Button_trendkr1" at 651,312 size 620x50; TextOff 'Кристализатор №1'
      on Release: ActivateScreen("Kristal_1", 0)
   Button "Button_trendkr2" at 651,367 size 620x50; TextOff 'Кристализатор №2'
      on Release: ActivateScreen("Kristal_2", 0)
   Button "Button_trendvo" at 651,422 size 620x50; TextOff 'Вакуумохладитель'
      on Release: ActivateScreen("VO", 0)

screen "VO" 1920x1080, template "Template_1"
   on GenerateScreen: SetTag("Tag_ScreenNumber", 7)
   TrendView "Trend view_1" at 0,51 size 1920x920

screen "settingsCommon" 1920x1080, template "Template_1"
   on GenerateScreen: SetTag("Tag_ScreenNumber", 4)
   Button "Buttonas_3" at 651,468 size 620x50; TextOff 'Общие настройки'
      on Release: ActivateScreen("settingsValue", 0)
   Button "Button_1123" at 651,300 size 620x50; TextOff 'Кристализатор №1'
      on Release: ActivateScreen("settingsKr1", 0)
   Button "Busadftton_1" at 651,356 size 620x50; TextOff 'Кристализатор №2'
      on Release: ActivateScreen("settingsKr2", 0)
   Button "Buttonas_2" at 651,412 size 620x50; TextOff 'Сип мойка'
      on Release: ActivateScreen("CIP", 0)

screen "CIP" 1920x1080, template "Template_1"
   TextField "Text field_2fsdf" at 877,654 size 114x25; Text 'Разрешение'
   TextField "Template_Text field_2" at 701,222 size 486x37; Text 'Управление режимами CIP мойки'
   SymbolicIOField "Symbolic I/O field_1" at 691,326 size 506x55; TextOff '0'; TextOn '1'; TextList "cipRegim"
      ProcessValue <- "Data_washing_cipRegim"
      ObjectEnable <- "WashingWork_DB_Run"
   Button "Button_9" at 956,387 size 241x55; TextOff 'Стоп'
      on Press: function_b14e0dd5("Data_washing_Stop", 0)
   Button "Button_111" at 691,387 size 241x55; TextOff 'Старт'
      on Press: function_b14e0dd5("Data_washing_Start", 0)
   Circle "Circle_1" at 783,468 size 48x48
      Appearance <- "Data_washing_readyGlobal"
   TextField "Text field_12cxvv" at 848,480 size 231x25; Text 'Готовность к включению'
   Circle "Circle_3" at 820,646 size 40x40
      Appearance <- "Data_ReadyCIP"
   Circle "Circle_4" at 820,589 size 40x40
      Appearance <- "Data_MAN_ON"
   TextField "asfasdf" at 877,597 size 214x25; Text 'Режим автоматический'
   TextField "Text field_1cip" at 877,540 size 155x25; Text 'Маршрут собран'
   Circle "Circle_2" at 820,532 size 40x40
      Appearance <- "Data_washing_readyRoute"

screen "settingsKr2" 1920x1080, template "Template_1"
   on GenerateScreen: SetTag("Tag_ScreenNumber", 9)
   TextField "Template_Text field_7" at 302,77 size 446x37; Text 'Параметры кристализации №2'
   TextField "Template_Text field_1" at 1209,77 size 360x37; Text 'Параметры мешалки №2'
   Group "Group_5" at 1048,147 size 594x341
   Group "Group" at 235,147 size 595x42
   Group "Group_2" at 235,199 size 595x42
   Group "Group_3" at 235,252 size 595x42
   Group "Group_4" at 235,304 size 595x42
   Circle "read_work_kr2" at 366,572 size 48x48
      Appearance <- "Data_Kr2_Ready_Work"
   TextField "Text field_12xcv" at 431,584 size 231x25; Text 'Готовность к включению'
   TextField "Text field_1asdf" at 460,644 size 155x25; Text 'Маршрут собран'
   Circle "ready_route_kr2" at 403,636 size 40x40
      Appearance <- "Data_Kr2_Ready_Route"
   Circle "Circle_11" at 403,693 size 40x40
      Appearance <- "Data_MAN_ON"
   TextField "Text field_3asdf" at 460,701 size 214x25; Text 'Режим автоматический'
   TextField "Text field_2asf" at 460,758 size 114x25; Text 'Разрешение'
   Circle "Circle_8" at 403,750 size 40x40
      Appearance <- "Data_ReadyKr2"
   SymbolicIOField "Symbolic I/O field_1" at 272,432 size 506x55; TextOff '0'; TextOn '1'; TextList "Kristal_Regim"
      ProcessValue <- "Data_Kr2_Regim"
      ObjectEnable <- "Kr_2_Work_Run"
   Button "Button_1bvn" at 272,493 size 241x55; TextOff 'Старт'
      on Press: function_b14e0dd5("Data_Kr2_Start", 0)
   Button "Button_2etd" at 537,493 size 241x55; TextOff 'Стоп'
      on Press: function_b14e0dd5("Data_Kr2_Stop", 0)
   IOField "IO Field_4" at 756,147 size 74x42; FormatPattern 999.9
      ProcessValue <- "Data_Kr2_TempFilling"
      ObjectEnable <- "Kr_2_Work_Run"
   TextField "Template_Text field_8" at 235,154 size 289x29; Text 'Температура наполнения, С°'
   IOField "IO Field_5" at 756,199 size 74x42; FormatPattern 999.9
      ProcessValue <- "Data_Kr2_TempKristal"
      ObjectEnable <- "Kr_2_Work_Run"
   TextField "Template_Text field_9" at 235,206 size 319x29; Text 'Температура кристализации, С°'
   IOField "IO Field_6" at 756,252 size 74x42; FormatPattern 9999
      ProcessValue <- "Data_Kr2_TimeKristal"
      ObjectEnable <- "Kr_2_Work_Run"
   TextField "Template_Text field_10" at 235,259 size 268x29; Text 'Время кристализации, мин'
   IOField "IO Field_7" at 756,304 size 74x42; FormatPattern 999
      ProcessValue <- "Kr_2_Work_LeftTimeMin"
   TextField "Template_Text field_11" at 235,311 size 296x29; Text 'До конца кристализации, мин'
   Button "Template_Button_1" at 1148,433 size 210x55; TextOff 'Старт мешалки'
      on Press: function_b14e0dd5("Data_Mixer2_Start", 0)
   Button "Template_Button_2" at 1369,433 size 210x55; TextOff 'Стоп мешалки'
      on Press: function_b14e0dd5("Data_Mixer2_Stop", 0)
   IOField "IO Field_15" at 1568,147 size 74x42; FormatPattern 999
      ProcessValue <- "Data_Mixer2_Power"
   TextField "Template_Text field_2" at 1048,154 size 217x29; Text 'Обороты мешалки, %'
   IOField "IO Field_1" at 1568,199 size 74x42; FormatPattern 9999
      ProcessValue <- "Data_Mixer2_TimeRight"
   TextField "Template_Text field_3" at 1048,206 size 288x29; Text 'Время вращения вправо, сек'
   IOField "IO Field_2" at 1568,252 size 74x42; FormatPattern 9999
      ProcessValue <- "Data_Mixer2_TimeLeft"
   TextField "Template_Text field_4" at 1048,259 size 276x29; Text 'Время вращения влево, сек'
   IOField "IO Field_3" at 1568,304 size 74x42; FormatPattern 9999
      ProcessValue <- "Data_Mixer2_TimePause"
   TextField "Template_Text field_5" at 1048,311 size 222x29; Text 'Время паузы мешалки'
   Group "Group_6" at 1048,147 size 594x42
   Group "Group_7" at 1048,199 size 594x42
   Group "Group_8" at 1048,252 size 594x42
   Group "Group_9" at 1048,304 size 594x42
   TextField "Template_Text field_6" at 1048,371 size 160x29; Text 'Режим мешалки'
   Button "Button_9" at 1392,358 size 118x55; TextOff '<< || >>'
      on Release: SetBit("Data_Mixer2_RegimBothSide")
      Appearance <- "Data_Mixer2_RegimBothSide"
   Button "Button_10" at 1524,358 size 118x55; TextOff '>>'
      on Release: ResetBit("Data_Mixer2_RegimBothSide")
      Appearance <- "Data_Mixer2_RegimBothSide"
   Group "Group_10" at 1148,433 size 431x55

screen "settingsValue" 1920x1080, template "Template_1"
   TextField "Template_Text field_2" at 783,170 size 258x37; Text 'Общие настройки'
   TextField "Template_Text field_3" at 554,285 size 288x54; Text 'Температура продукта после вакуумного охладителя, C°'
   IOField "IO Field_2" at 1149,291 size 74x42; FormatPattern 999.9
      ProcessValue <- "Data_Reg_01RV01_Sp"
   TextField "Template_Text field_8" at 554,238 size 303x29; Text 'Уровень вакуумохладителя, %'
   IOField "IO Field_4" at 1149,231 size 74x42; FormatPattern 999.9
      ProcessValue <- "Data_Reg_M7_1_Sp"
   TextField "Template_Text field_1" at 554,360 size 390x29; Text 'Мощность насоса M7_2 на продукте, %'
   IOField "IO Field_1" at 1149,353 size 74x42; FormatPattern 999
      ProcessValue <- "Data_Power_7_2"
   TextField "Template_Text field_4" at 554,415 size 359x29; Text 'Мощность насоса M7_2 на мойке, %'
   IOField "IO Field_3" at 1149,408 size 74x42; FormatPattern 999
      ProcessValue <- "Data_Power_7_2_CIP"
   TextField "Template_Text field_5" at 554,478 size 385x29; Text 'Блокировка разрешение на включение'
   SymbolicIOField "Symbolic I/O field_1" at 1040,471 size 182x42; TextOff '0'; TextOn '1'; TextList "on/off"; Authorization "Operate"
      ProcessValue <- "Data_EnableReady"
*)

(* ===== HMI "HMI_RT_1" =====

ScreenModuleEditorView "V7_31" 640x480
   SymbolLibrary "Symbol library_9" at 10,10 size 50x42
*)

(* ===== HMI "HMI_RT_1" =====

ScreenModuleEditorView "V7_31" 640x480
   SymbolLibrary "Symbol library_9" at 126,71 size 50x42
      Appearance <- "Km1"
   SymbolLibrary "Symbol library_1" at 126,71 size 50x42
      Visibility <- "Err"
*)

(* ===== HMI "HMI_RT_1" =====

ScreenModuleEditorView "М7_4" 640x480
   SymbolLibrary "Symbol library_13" at 254,88 size 42x50
      Appearance <- "Km1"
   SymbolLibrary "Symbol library_1" at 254,88 size 42x50
      Visibility <- "Err"
*)

(* ===== HMI "HMI_RT_1" =====

ScreenModuleEditorView "M7_1" 640x480
   SymbolLibrary "Symbol library_33" at 10,10 size 88x65
      Appearance <- "Km1"
   SymbolLibrary "Symbol library_1" at 10,10 size 88x65
      Visibility <- "Err"
*)

(* ===== HMI "HMI_RT_1" =====

ScreenModuleEditorView "M7_2" 640x480
   SymbolLibrary "Symbol library_60" at 123,72 size 77x54
      Appearance <- "Km1"
   SymbolLibrary "Symbol library_1" at 123,72 size 77x54
      Visibility <- "Err"
*)

(* ===== HMI "HMI_RT_1" =====

ScreenModuleEditorView "M1_2" 640x480
   SymbolLibrary "Symbol library_62" at 10,10 size 60x51
      Appearance <- "Km1"
   SymbolLibrary "Symbol library_1" at 10,10 size 60x51
      Visibility <- "Err"
*)

(* ===== HMI "HMI_RT_1" =====

ScreenModuleEditorView "M1_1" 640x480
   SymbolLibrary "Symbol library_166" at 42,50 size 53x69
      Appearance <- "Km1"
   SymbolLibrary "Symbol library_1" at 42,50 size 53x69
      Visibility <- "Err"
*)

(* ===== HMI "HMI_RT_1" =====

ScreenModuleEditorView "V7_2" 640x480
   SymbolLibrary "Symbol library_39" at 10,10 size 26x35
      Appearance <- "Km1"
   SymbolLibrary "Symbol library_1" at 10,10 size 26x35
      Visibility <- "Err"
*)

(* ===== HMI "HMI_RT_1" =====

ScreenModuleEditorView "M_3" 640x480
   SymbolLibrary "Symbol library_155" at 10,10 size 60x51
      Appearance <- "Km1"
   SymbolLibrary "Symbol library_1" at 10,10 size 60x51
      Visibility <- "Err"
*)

(* ===== HMI "HMI_RT_1" =====

ScreenModuleEditorView "V1_7" 640x480
   SymbolLibrary "Symbol library_49" at 10,10 size 35x26
      Appearance <- "Km1"
   SymbolLibrary "Symbol library_1" at 10,10 size 35x26
      Visibility <- "Err"
*)

(* ===== HMI "HMI_RT_1" =====

ScreenModuleEditorView "RV01" 640x480
   SymbolLibrary "Symbol library_125" at 10,10 size 51x64
   SymbolLibrary "Symbol library_1" at 10,10 size 51x64
      Appearance <- "Px"
*)

(* ===== HMI "HMI_RT_1" =====

ScreenModuleEditorView "M7_21" 640x480
   SymbolLibrary "Symbol library_28" at 10,10 size 77x60
      Appearance <- "Km1"
   SymbolLibrary "Symbol library_1" at 10,10 size 77x60
      Visibility <- "Err"
*)